Fanuc KAREL source: kt00548.KL

-- PROVISIONAL review KL for V770-1; original PC SHA256 d54ac1a2477a3666c37ba6d1a1e1979ca04d254a0009af860ab69118826ee10d
-- Incomplete behavior may be omitted. Consult companion uncertainty JSON. Do not deploy.
PROGRAM KT00548
%NOLOCKGROUP
VAR
  OUT : BOOLEAN
-- UNRESOLVED_DECL P1 type=000199
-- UNRESOLVED_DECL P2 type=000199
BEGIN
  -- UNRESOLVED_PC offsets 5-38; opcodes 49,7E,49,7E,AC,23
  -- UNRESOLVED_PC offsets 43-47; opcodes 7F
END KT00548
